# EPICS substitutions: viocs/ts_ps/ts_psApp/Db/ch.substitutions
file "db/individual.db" {
    pattern { family, pos }
        { "CH", "01" }
        { "CH", "02" }
        { "CH", "03" }
        { "CH", "04" }
}
